INTERFACE I_ServerResponseHeaderAccessor

METHOD PUBLIC UpdateResponseWithAccepted
VAR_INPUT
	Response : I_ServerResponse;
END_VAR
END_METHOD

METHOD PUBLIC UpdateResponseWithBusy
VAR_INPUT
	Response : I_ServerResponse;
END_VAR
END_METHOD

METHOD PUBLIC UpdateResponseWithError
VAR_INPUT
	Response : I_ServerResponse;
	Message : T_MAXSTRING;
END_VAR
END_METHOD

METHOD PUBLIC UpdateResponseWithPending
VAR_INPUT
	Response : I_ServerResponse;
	ResponseId : T_MAXSTRING;
	RetryDelayInMs : UDINT;
END_VAR
END_METHOD

METHOD PUBLIC UpdateResponseWithSuccess
VAR_INPUT
	Response : I_ServerResponse;
END_VAR
END_METHOD

END_INTERFACE

(* stored: Version 1.1.0.1, ProductVersion 3.1.4024.12
   Itf I_ServerResponseHeaderAccessor: Id {53bef890-c057-0df6-052a-6ae563d65901}
   Method UpdateResponseWithAccepted: Id {c20aed84-d249-0855-3097-3219546eee7e}
   Method UpdateResponseWithBusy: Id {f4a0c291-b7d7-09e6-0cb5-c8e319701f0f}
   Method UpdateResponseWithError: Id {1e97ceb8-7123-0088-09fe-83219ced09a7}
   Method UpdateResponseWithPending: Id {a5368b50-802f-04a8-3040-2d1aa4dde5d5}
   Method UpdateResponseWithSuccess: Id {5e4264a1-461e-03fb-01ec-3a802132c53d} *)
